// Mitsubishi GX Works2 project: INC, DEC   PLC: Q02/Q02H

PROGRAM MAIN
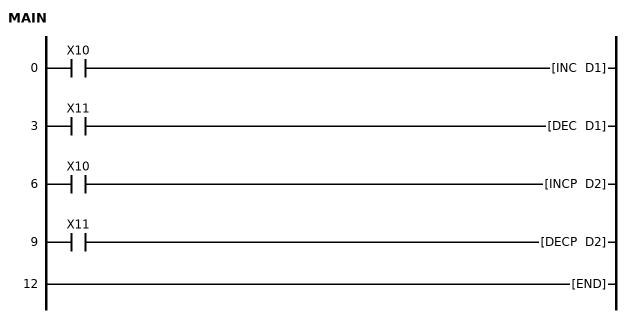
0     LD      X10
      INC     D1
3     LD      X11
      DEC     D1
6     LD      X10
      INCP    D2
9     LD      X11
      DECP    D2
12    END
END_PROGRAM

PROGRAM MAIN1
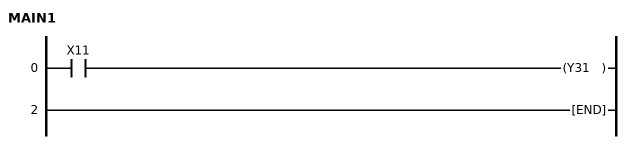
0     LD      X11
      OUT     Y31
2     END
END_PROGRAM
